// TwinCAT 3 PLC project Data
// Title: Data
// Company: TomasRompotl
// ProjectVersion: 0.0.1
// ProgramVersion: 3.1.4024.0
// libraries:
//   Base Interfaces,newest,System
//   Strings, * (TomasRompotl)
//   Tc2_System, * (Beckhoff Automation GmbH)
//   Tc2_Utilities, * (Beckhoff Automation GmbH)
// project tree:
//   Comparison/ CompareAnyType.TcPOU, ComparisonOperator.TcDUT, DataEquals.TcPOU, IsEqualAnyType.TcPOU, IsGreaterThanAnyType.TcPOU, IsGreaterThanOrEqualAnyType.TcPOU (not stored), IsLessThanAnyType.TcPOU, IsLessThanOrEqualAnyType.TcPOU, IsNotEqualAnyType.TcPOU
//   Manipulate/ ClearData.TcPOU, ClearDataAnyType.TcPOU (not stored), ShiftDataLeft.TcPOU, ShiftDataRight.TcPOU, Swap.TcPOU, SwapByPointer.TcPOU
//   QuickSort/ PartitionREAL.TcPOU (not stored), QuickSortREAL.TcPOU (not stored)
//   Sort/ SortOrder.TcTLEO, SortAnything.TcPOU (not stored), _Partition.TcPOU, _QuickSort.TcPOU
//   TableSerialization/ TableDeserializer.TcPOU, TableSerializationParameters.TcGVL (not stored), TableSerializer.TcPOU
//   Version/ Global_Version.TcGVL
// (motion and I/O tree: see PLC project types)
// real-time tasks:
//   TASK BindingTestTask: cycle T#10ms, priority 20, ADS port 350
//   TASK PlcTask: cycle T#10ms, priority 21, ADS port 351
//   TASK PlcTask1: cycle T#10ms, priority 22, ADS port 352
//   TASK PlcTask2: cycle T#10ms, priority 23, ADS port 353

// ---- Comparison/ComparisonOperator.TcDUT
{attribute 'qualified_only'}
{attribute 'strict'}
TYPE ComparisonOperator :
(
	Equal,
	NotEqual,
	LessThan,
	LessThenOrEqual,
	GreaterThan,
	GreaterThanOrEqual
);
END_TYPE

// ---- Sort/SortOrder.TcTLEO
{attribute 'qualified_only'}
{attribute 'strict'}
TYPE SortOrder :
(
	ASCENDING,
	DESCENDING
);
END_TYPE

// ---- Version/Global_Version.TcGVL
{attribute 'TcGenerated'}
{attribute 'no-analysis'}
{attribute 'linkalways'}
// This function has been automatically generated from the project information.
VAR_GLOBAL CONSTANT
	{attribute 'const_non_replaced'}
	stLibVersion_Data : ST_LibVersion := (iMajor := 0, iMinor := 0, iBuild := 1, iRevision := 0, nFlags := 0, sVersion := '0.0.1');
END_VAR

// ---- Comparison/CompareAnyType.TcPOU
FUNCTION CompareAnyType : BOOL
VAR_INPUT
	a					: __SYSTEM.AnyType; // a and b have to be same type
	is					: ComparisonOperator;
	b					: __SYSTEM.AnyType; // a and b have to be same type
END_VAR

CASE is OF
	ComparisonOperator.Equal:
		CompareAnyType := IsEqualAnyType(a, b);
	ComparisonOperator.NotEqual:
		CompareAnyType := IsNotEqualAnyType(a, b);
	ComparisonOperator.LessThan:
		CompareAnyType := IsLessThanAnyType(a, b);
	ComparisonOperator.LessThanOrEqual:
		CompareAnyType := IsLessThanOrEqualAnyType(a, b);
	ComparisonOperator.GreaterThan:
		CompareAnyType := IsGreaterThanAnyType(a, b);
	ComparisonOperator.GreaterThanOrEqual:
		CompareAnyType := IsGreaterThanOrEqualAnyType(a, b);
END_CASE

END_FUNCTION

// ---- Comparison/IsEqualAnyType.TcPOU
FUNCTION IsEqualAnyType : BOOL
VAR_INPUT
	a					: __SYSTEM.AnyType; // A and B have to be same type
	b					: __SYSTEM.AnyType; // A and B have to be same type
END_VAR

IF a.TypeClass <> b.TypeClass THEN
	RETURN;
END_IF

IsEqualAnyType := MEMCMP(a.pValue, b.pValue, TO_UDINT(a.diSize)) = 0;

END_FUNCTION

// ---- Comparison/IsNotEqualAnyType.TcPOU
FUNCTION IsNotEqualAnyType : BOOL
VAR_INPUT
	a					: __SYSTEM.AnyType; // A and B have to be same type
	b					: __SYSTEM.AnyType; // A and B have to be same type
END_VAR

IsNotEqualAnyType := NOT IsEqualAnyType(a, b);

END_FUNCTION

// ---- Comparison/IsLessThanAnyType.TcPOU
FUNCTION IsLessThanAnyType : BOOL
VAR_INPUT
	a					: __SYSTEM.AnyType; // A and B have to be same type
	b					: __SYSTEM.AnyType; // A and B have to be same type
END_VAR

IF a.TypeClass <> b.TypeClass THEN
	RETURN;
END_IF

CASE UDINT_TO_INT(a.TypeClass) OF
    IBaseLibrary.TypeClass.TYPE_BOOL :
        IsLessThanAnyType := PBOOL_TO_BOOL(a.pValue) < PBOOL_TO_BOOL(b.pValue);
    IBaseLibrary.TypeClass.TYPE_BIT :
        IsLessThanAnyType := BYTE_TO_BIT(a.pValue^) < BYTE_TO_BIT(b.pValue^);
    IBaseLibrary.TypeClass.TYPE_BYTE :
        IsLessThanAnyType := a.pValue^ < b.pValue^;
    IBaseLibrary.TypeClass.TYPE_WORD :
        IsLessThanAnyType := PWORD_TO_WORD(a.pValue) < PWORD_TO_WORD(b.pValue);
    IBaseLibrary.TypeClass.TYPE_DWORD :
        IsLessThanAnyType := PDWORD_TO_DWORD(a.pValue) < PDWORD_TO_DWORD(b.pValue);
    IBaseLibrary.TypeClass.TYPE_LWORD :
        IsLessThanAnyType := PLWORD_TO_LWORD(a.pValue) < PLWORD_TO_LWORD(b.pValue);
    IBaseLibrary.TypeClass.TYPE_SINT :
        IsLessThanAnyType := PSINT_TO_SINT(a.pValue) < PSINT_TO_SINT(b.pValue);
    IBaseLibrary.TypeClass.TYPE_INT :
        IsLessThanAnyType := PINT_TO_INT(a.pValue) < PINT_TO_INT(b.pValue);
    IBaseLibrary.TypeClass.TYPE_DINT :
        IsLessThanAnyType := PDINT_TO_DINT(a.pValue) < PDINT_TO_DINT(b.pValue);
    IBaseLibrary.TypeClass.TYPE_LINT :
        IsLessThanAnyType := PLINT_TO_LINT(a.pValue) < PLINT_TO_LINT(b.pValue);
    IBaseLibrary.TypeClass.TYPE_USINT :
        IsLessThanAnyType := PUSINT_TO_USINT(a.pValue) < PUSINT_TO_USINT(b.pValue);
    IBaseLibrary.TypeClass.TYPE_UINT :
        IsLessThanAnyType := PUINT_TO_UINT(a.pValue) < PUINT_TO_UINT(b.pValue);
    IBaseLibrary.TypeClass.TYPE_UDINT :
        IsLessThanAnyType := PUDINT_TO_UDINT(a.pValue) < PUDINT_TO_UDINT(b.pValue);
    IBaseLibrary.TypeClass.TYPE_ULINT :
        IsLessThanAnyType := PULINT_TO_ULINT(a.pValue) < PULINT_TO_ULINT(b.pValue);
    IBaseLibrary.TypeClass.TYPE_REAL :
        IsLessThanAnyType := PREAL_TO_REAL(a.pValue) < PREAL_TO_REAL(b.pValue);
    IBaseLibrary.TypeClass.TYPE_LREAL :
        IsLessThanAnyType := PLREAL_TO_LREAL(a.pValue) < PLREAL_TO_LREAL(b.pValue);
    IBaseLibrary.TypeClass.TYPE_STRING :
        IsLessThanAnyType := PSTRING_TO_STRING(a.pValue) < PSTRING_TO_STRING(b.pValue);
    IBaseLibrary.TypeClass.TYPE_TIME :
        IsLessThanAnyType := PTIME_TO_TIME(a.pValue) < PTIME_TO_TIME(b.pValue);
    IBaseLibrary.TypeClass.TYPE_DATE :
        IsLessThanAnyType := PDATE_TO_DATE(a.pValue) < PDATE_TO_DATE(b.pValue);
    IBaseLibrary.TypeClass.TYPE_DATEANDTIME :
        IsLessThanAnyType := PDT_TO_DT(a.pValue) < PDT_TO_DT(b.pValue);
    IBaseLibrary.TypeClass.TYPE_TIMEOFDAY :
        IsLessThanAnyType := PTOD_TO_TOD(a.pValue) < PTOD_TO_TOD(b.pValue);
    IBaseLibrary.TypeClass.TYPE_POINTER :
        IsLessThanAnyType := a.pValue < b.pValue;
    IBaseLibrary.TypeClass.TYPE_LTIME :
        IsLessThanAnyType := PLTIME_TO_LTIME(a.pValue) < PLTIME_TO_LTIME(b.pValue);
	ELSE
		RETURN;
END_CASE

END_FUNCTION

// ---- Comparison/IsLessThanOrEqualAnyType.TcPOU
FUNCTION IsLessThanOrEqualAnyType : BOOL
VAR_INPUT
	a					: __SYSTEM.AnyType; // A and B have to be same type
	b					: __SYSTEM.AnyType; // A and B have to be same type
END_VAR

IsLessThanOrEqualAnyType := NOT IsGreaterThanAnyType(a, b);

END_FUNCTION

// ---- Comparison/IsGreaterThanAnyType.TcPOU
FUNCTION IsGreaterThanAnyType : BOOL
VAR_INPUT
	a					: __SYSTEM.AnyType; // A and B have to be same type
	b					: __SYSTEM.AnyType; // A and B have to be same type
END_VAR

IF a.TypeClass <> b.TypeClass THEN
	RETURN;
END_IF

CASE UDINT_TO_INT(a.TypeClass) OF
    IBaseLibrary.TypeClass.TYPE_BOOL :
        IsGreaterThanAnyType := PBOOL_TO_BOOL(a.pValue) > PBOOL_TO_BOOL(b.pValue);
    IBaseLibrary.TypeClass.TYPE_BIT :
        IsGreaterThanAnyType := BYTE_TO_BIT(a.pValue^) > BYTE_TO_BIT(b.pValue^);
    IBaseLibrary.TypeClass.TYPE_BYTE :
        IsGreaterThanAnyType := a.pValue^ > b.pValue^;
    IBaseLibrary.TypeClass.TYPE_WORD :
        IsGreaterThanAnyType := PWORD_TO_WORD(a.pValue) > PWORD_TO_WORD(b.pValue);
    IBaseLibrary.TypeClass.TYPE_DWORD :
        IsGreaterThanAnyType := PDWORD_TO_DWORD(a.pValue) > PDWORD_TO_DWORD(b.pValue);
    IBaseLibrary.TypeClass.TYPE_LWORD :
        IsGreaterThanAnyType := PLWORD_TO_LWORD(a.pValue) > PLWORD_TO_LWORD(b.pValue);
    IBaseLibrary.TypeClass.TYPE_SINT :
        IsGreaterThanAnyType := PSINT_TO_SINT(a.pValue) > PSINT_TO_SINT(b.pValue);
    IBaseLibrary.TypeClass.TYPE_INT :
        IsGreaterThanAnyType := PINT_TO_INT(a.pValue) > PINT_TO_INT(b.pValue);
    IBaseLibrary.TypeClass.TYPE_DINT :
        IsGreaterThanAnyType := PDINT_TO_DINT(a.pValue) > PDINT_TO_DINT(b.pValue);
    IBaseLibrary.TypeClass.TYPE_LINT :
        IsGreaterThanAnyType := PLINT_TO_LINT(a.pValue) > PLINT_TO_LINT(b.pValue);
    IBaseLibrary.TypeClass.TYPE_USINT :
        IsGreaterThanAnyType := PUSINT_TO_USINT(a.pValue) > PUSINT_TO_USINT(b.pValue);
    IBaseLibrary.TypeClass.TYPE_UINT :
        IsGreaterThanAnyType := PUINT_TO_UINT(a.pValue) > PUINT_TO_UINT(b.pValue);
    IBaseLibrary.TypeClass.TYPE_UDINT :
        IsGreaterThanAnyType := PUDINT_TO_UDINT(a.pValue) > PUDINT_TO_UDINT(b.pValue);
    IBaseLibrary.TypeClass.TYPE_ULINT :
        IsGreaterThanAnyType := PULINT_TO_ULINT(a.pValue) > PULINT_TO_ULINT(b.pValue);
    IBaseLibrary.TypeClass.TYPE_REAL :
        IsGreaterThanAnyType := PREAL_TO_REAL(a.pValue) > PREAL_TO_REAL(b.pValue);
    IBaseLibrary.TypeClass.TYPE_LREAL :
        IsGreaterThanAnyType := PLREAL_TO_LREAL(a.pValue) > PLREAL_TO_LREAL(b.pValue);
    IBaseLibrary.TypeClass.TYPE_STRING :
        IsGreaterThanAnyType := PSTRING_TO_STRING(a.pValue) > PSTRING_TO_STRING(b.pValue);
    IBaseLibrary.TypeClass.TYPE_TIME :
        IsGreaterThanAnyType := PTIME_TO_TIME(a.pValue) > PTIME_TO_TIME(b.pValue);
    IBaseLibrary.TypeClass.TYPE_DATE :
        IsGreaterThanAnyType := PDATE_TO_DATE(a.pValue) > PDATE_TO_DATE(b.pValue);
    IBaseLibrary.TypeClass.TYPE_DATEANDTIME :
        IsGreaterThanAnyType := PDT_TO_DT(a.pValue) > PDT_TO_DT(b.pValue);
    IBaseLibrary.TypeClass.TYPE_TIMEOFDAY :
        IsGreaterThanAnyType := PTOD_TO_TOD(a.pValue) > PTOD_TO_TOD(b.pValue);
    IBaseLibrary.TypeClass.TYPE_POINTER :
        IsGreaterThanAnyType := a.pValue > b.pValue;
    IBaseLibrary.TypeClass.TYPE_LTIME :
        IsGreaterThanAnyType := PLTIME_TO_LTIME(a.pValue) > PLTIME_TO_LTIME(b.pValue);
	ELSE
		RETURN;
END_CASE

END_FUNCTION

// ---- Comparison/DataEquals.TcPOU
FUNCTION DataEquals : BOOL
VAR_INPUT
	a : ANY;
	b : ANY;
END_VAR
VAR
END_VAR

IF (a.diSize <> b.diSize) THEN
	RETURN;
END_IF

DataEquals := MEMCMP(pBuf1 := a.pValue, pBuf2 := b.pValue, n := a.diSize) = 0;

END_FUNCTION

// ---- Manipulate/ClearData.TcPOU
FUNCTION ClearData : BOOL
VAR_INPUT
	data : ANY;
END_VAR

MEMSET(destAddr := data.pValue, fillByte := 0, n := TO_UDINT(data.diSize));

END_FUNCTION

// ---- Manipulate/ShiftDataLeft.TcPOU
// Shift data from end to begin
FUNCTION ShiftDataLeft : BOOL
VAR_INPUT
	data : ANY;
	byteCount : UDINT; // How far to the left are shifted
END_VAR

MEMMOVE(destAddr := data.pValue, srcAddr := data.pValue + byteCount, n := TO_UDINT(data.diSize) - byteCount);
MEMSET(destAddr := data.pValue + TO_UDINT(data.diSize) - byteCount, fillByte := 0, n := byteCount);

END_FUNCTION

// ---- Manipulate/ShiftDataRight.TcPOU
// Shift data from end to begin
FUNCTION ShiftDataRight : BOOL
VAR_INPUT
	data : ANY;
	byteCount : UDINT; // How far to the right are shifted
END_VAR

MEMMOVE(destAddr := data.pValue + byteCount, srcAddr := data.pValue, data.diSize - byteCount);
MEMSET(destAddr := data.pValue, fillByte := 0, n := byteCount);

END_FUNCTION

// ---- Manipulate/Swap.TcPOU
// Swaps values of two variables
FUNCTION Swap
VAR_INPUT
	a : ANY;
	b : ANY;
END_VAR
VAR
	temp : POINTER TO BYTE;
END_VAR

temp := __NEW(BYTE, a.diSize);

MEMCPY(temp, a.pValue, a.diSize);
MEMCPY(a.pValue, b.pValue, a.diSize);
MEMCPY(b.pValue, temp, a.diSize);

__DELETE(temp);

END_FUNCTION

// ---- Manipulate/SwapByPointer.TcPOU
// Swaps values of two variables
FUNCTION SwapByPointer
VAR_INPUT
	a : POINTER TO BYTE;
	b : POINTER TO BYTE;
	length : DINT;
END_VAR
VAR
	temp : POINTER TO BYTE;
END_VAR

temp := __NEW(BYTE, TO_UDINT(length));

MEMCPY(temp, a, TO_UDINT(length));
MEMCPY(a, b, TO_UDINT(length));
MEMCPY(b, temp, TO_UDINT(length));

__DELETE(temp);

END_FUNCTION

// ---- Sort/_Partition.TcPOU
// Function used in QuickSort
FUNCTION _Partition : DINT
VAR_INPUT
	arr					: __SYSTEM.AnyType;
	firstElement		: __SYSTEM.AnyType;
	sortBy				: __SYSTEM.AnyType;
	memberOffset		: DWORD;
	startIndex			: DINT; // Starting comparision index
	endIndex			: DINT; // Ending comparision index
	order 				: SortOrder;
END_VAR
VAR
	pivot				: POINTER TO BYTE; // Compared number
	leftwall			: DINT; // New pivot location
	iterator			: DINT; // For iterator variable
	iterAdr				: POINTER TO BYTE;
	compA				: __SYSTEM.AnyType := sortBy; // get data of compared variable
	compB				: __SYSTEM.AnyType := sortBy;
END_VAR

pivot := arr.pValue + firstElement.diSize * endIndex;
leftwall := startIndex;

FOR iterator := startIndex TO endIndex - 1 DO

	iterAdr := arr.pValue + firstElement.diSize * iterator;
	
	compA.pValue := iterAdr + memberOffset; // data of compared variable stays the same, just point to other value
	compB.pValue := pivot + memberOffset;
	
	CASE order OF
		SortOrder.ASCENDING:
			IF (IsLessThanOrEqualAnyType(compA, compB)) THEN

				SwapByAddr(iterAdr, arr.pValue + firstElement.diSize * leftwall, firstElement.diSize);
				leftwall := leftwall + 1;
			END_IF
		SortOrder.DESCENDING:
			IF (IsGreaterThanOrEqualAnyType(compA, compB)) THEN

				SwapByAddr(iterAdr, arr.pValue + firstElement.diSize * leftwall, firstElement.diSize);
				leftwall := leftwall + 1;
			END_IF
	END_CASE
END_FOR

SwapByAddr(arr.pValue + firstElement.diSize * leftwall, pivot, firstElement.diSize);

_Partition := leftwall;

END_FUNCTION

// ---- Sort/_QuickSort.TcPOU

FUNCTION _QuickSort
VAR_INPUT
	Arr					: __SYSTEM.AnyType;
	FirstElement		: __SYSTEM.AnyType;
	SortBy				: __SYSTEM.AnyType;
	MemberOffset		: DWORD;
	StartIndex			: DINT; // Start index
	EndIndex			: DINT; // End index
	Order 				: SortOrder;
END_VAR
VAR 
	PivotIndex			: DINT; // Partitioning point
END_VAR


IF StartIndex < EndIndex THEN

	PivotIndex := _Partition(Arr, FirstElement, SortBy, MemberOffset, StartIndex, EndIndex, Order);
	_QuickSort(Arr, FirstElement, SortBy, MemberOffset, StartIndex, PivotIndex - 1, Order);
	_QuickSort(Arr, FirstElement, SortBy, MemberOffset, PivotIndex + 1, EndIndex, Order);
END_IF

END_FUNCTION

// ---- TableSerialization/TableDeserializer.TcPOU
FUNCTION_BLOCK TableDeserializer
VAR
	_DataString : POINTER TO STRING;
	dataLength : DINT;
	rowDefinition : __SYSTEM.AnyType;
	_RowCount : DINT;
	_ColumnDefinitionBuffer : ARRAY[0..MaxColumnCount - 1] OF __SYSTEM.AnyType;
	_ColumnNameBuffer : ARRAY[0..MaxColumnCount - 1] OF T_MaxString;
	columnNamesOutput : __SYSTEM.AnyType;
	definedColumns : INT;

	_Separator : STRING := ',';
	_NewLine : STRING := '$N'; // Default is Windows newline.
	_DecimalSeparator : STRING := '.';
END_VAR
VAR CONSTANT
	MaxColumnCount : INT := TableSerializationParameters.DeserializerMaxColumns;
	DefaultDecimalSeparator : STRING := '.';
END_VAR

{attribute 'monitoring' := 'call'}
PROPERTY DataString : POINTER TO STRING
GET
DataString := _DataString;
END_GET
SET
_DataString := DataString;
END_SET
END_PROPERTY

{attribute 'monitoring' := 'call'}
PROPERTY DecimalSeparator : STRING
GET
DecimalSeparator := _DecimalSeparator;
END_GET
SET
_DecimalSeparator := DecimalSeparator;
END_SET
END_PROPERTY

METHOD DefineColumnNamesOutput : REFERENCE TO TableDeserializer
VAR_INPUT
	columnNames : ANY; 
END_VAR
columnNamesOutput := columnNames;

DefineColumnNamesOutput REF= THIS^;
END_METHOD

METHOD DefineNextColumn : REFERENCE TO TableDeserializer
VAR_INPUT
	columnInFirstRow : ANY; 
END_VAR
IF (definedColumns < MaxColumnCount) THEN
	_ColumnDefinitionBuffer[definedColumns] := columnInFirstRow;
	definedColumns := definedColumns + 1;
END_IF

DefineNextColumn REF= THIS^;
END_METHOD

METHOD DefineRow : REFERENCE TO TableDeserializer
VAR_INPUT
	firstRow : ANY;
END_VAR
rowDefinition := firstRow;

DefineRow REF= THIS^;
END_METHOD

METHOD Deserialize : DINT
VAR_INPUT
	includingHeader : BOOL;
END_VAR
VAR
	caret : DINT;
END_VAR
dataLength := LEN2(dataString);
IF (includingHeader) THEN
	caret := ReadHeader();
END_IF
caret := ReadAllRows(caret);

Deserialize := caret;
END_METHOD

{attribute 'monitoring' := 'call'}
PROPERTY NewLine : STRING
GET
NewLine := _NewLine;
END_GET
SET
_NewLine := NewLine;
END_SET
END_PROPERTY

METHOD PRIVATE ReadAllRows : DINT
VAR_INPUT
	startCaret : DINT;
END_VAR
VAR
	caret : DINT;
	i : DINT;
END_VAR
caret := startCaret;

FOR i := 0 TO _RowCount - 1 DO
	IF (caret >= dataLength) THEN
		EXIT;
	END_IF
	caret := ReadRow(i, caret);
END_FOR

ReadAllRows := caret;
END_METHOD

METHOD PRIVATE ReadHeader : DINT
VAR
	i : DINT;
	
	caret : DINT;
	lineEnd : DINT;
	cellLength : DINT;
	
	cell : T_MaxString;
END_VAR
ClearData(_ColumnNameBuffer);

lineEnd := FIND2(pSrcString := _DataString, pFindString := ADR(_NewLine));
IF (lineEnd = 0) THEN
	lineEnd := dataLength;
END_IF

FOR i := 0 TO definedColumns - 1 DO
	cellLength := FIND2(pSrcString := _DataString + caret, pFindString := ADR(_Separator));
	IF (caret + cellLength > lineEnd) THEN
		cellLength := lineEnd - caret;
	END_IF
	IF (cellLength = 0) THEN
		cellLength := lineEnd;
	END_IF

	MEMSET(destAddr := ADR(cell), fillByte := 0, n := SIZEOF(cell));
	MEMCPY(destAddr := ADR(cell), srcAddr := _DataString + caret, n := MIN(SIZEOF(cell) - 1, cellLength - 1));
	StringToAny(cell, _ColumnNameBuffer[i]);
	
	IF (cellLength = dataLength) THEN
		caret := lineEnd;
	ELSIF (cellLength = lineEnd) THEN
		caret := lineEnd;
	ELSE
		caret := caret + cellLength;
	END_IF
END_FOR

MEMCPY(
	destAddr := columnNamesOutput.pValue,
	srcAddr := ADR(_ColumnNameBuffer),
	n := MIN(columnNamesOutput.diSize, SIZEOF(_ColumnNameBuffer))
);

ReadHeader := caret;
END_METHOD

METHOD PRIVATE ReadRow : DINT
VAR_INPUT
	row : DINT;
	startCaret : DINT;
END_VAR
VAR
	i : DINT;
	
	caret : DINT;
	lineLength : DINT;
	cellLength : DINT;
	
	cell : T_MaxString;
	
	tableCell : __SYSTEM.AnyType;
END_VAR
caret := startCaret;

lineLength := FIND2(pSrcString := _DataString + caret, pFindString := ADR(_NewLine));
IF (lineLength = 0) THEN
	lineLength := dataLength;
END_IF

FOR i := 0 TO definedColumns - 1 DO
  IF (caret >= dataLength) THEN
		EXIT;
	END_IF
	cellLength := FIND2(pSrcString := _DataString + caret, pFindString := ADR(_Separator));
	IF (cellLength = 0 OR caret + cellLength > startCaret + lineLength) THEN
		cellLength := lineLength + startCaret - caret;
	END_IF
	IF (cellLength = 0) THEN
		caret := dataLength;
		EXIT;
	END_IF

	ClearData(cell);
	MEMCPY(destAddr := ADR(cell), srcAddr := _DataString + caret, n := MIN(SIZEOF(cell) - 1, cellLength - 1));
	tableCell := _ColumnDefinitionBuffer[i];
	tableCell.pValue := tableCell.pValue + rowDefinition.diSize * row;
	CASE tableCell.TypeClass OF
		TYPE_REAL, TYPE_LREAL:
			ReplaceString(cell, _DecimalSeparator, DefaultDecimalSeparator);
	END_CASE
	StringToAnyType(cell, tableCell);
	
	IF (cellLength = dataLength) THEN
		caret := startCaret + lineLength;
	ELSIF (cellLength = lineLength) THEN
		caret := startCaret + lineLength;
	ELSE
		caret := caret + cellLength;
	END_IF
END_FOR

ReadRow := caret;
END_METHOD

{attribute 'monitoring' := 'call'}
PROPERTY RowCount : DINT
GET
RowCount := _RowCount;
END_GET
SET
_RowCount := RowCount;
END_SET
END_PROPERTY

{attribute 'monitoring' := 'call'}
PROPERTY Separator : STRING
GET
Separator := _Separator;
END_GET
SET
_Separator := Separator;
END_SET
END_PROPERTY

END_FUNCTION_BLOCK

// ---- TableSerialization/TableSerializer.TcPOU
FUNCTION_BLOCK TableSerializer
VAR
	_StringBuilder : REFERENCE TO StringBuilderExtBuffer;
	
	rowDefinition : __SYSTEM.AnyType;
	_RowCount : DINT;
	_ColumnDefinitionBuffer : ARRAY[0..MaxColumnCount - 1] OF __SYSTEM.AnyType;
	_ColumnNameBuffer : ARRAY[0..MaxColumnCount - 1] OF T_MaxString;
	definedColumns : INT;
	
	_Separator : STRING := ','; // Default separator ';' is compatible with european decimal separator '.'.
	_NewLine : STRING := '$N'; // Default is Windows newline.
	_DecimalSeparator : STRING := '.';
END_VAR
VAR CONSTANT
	MaxColumnCount : INT := TableSerializationParameters.SerializerMaxColumns;
	DefaultDecimalSeparator : STRING := '.';
END_VAR

METHOD PRIVATE AddColumnHeader
VAR
	column : INT;
END_VAR
FOR column := 0 TO definedColumns - 1 DO
	IF (column > 0) THEN
		_StringBuilder.Append(_Separator);
	END_IF
	
	_StringBuilder.Append(_ColumnNameBuffer[column]);
END_FOR
END_METHOD

METHOD PRIVATE AddLine
VAR_INPUT
	rowIndex : DINT;
END_VAR
VAR
	column : INT;
	currentData : __SYSTEM.AnyType;
	converted : T_MaxString;
END_VAR
FOR column := 0 TO definedColumns - 1 DO
	IF (column > 0) THEN
		_StringBuilder.Append(_Separator);
	END_IF
	
	currentData := _ColumnDefinitionBuffer[column];
	currentData.pValue := rowDefinition.pValue + (rowDefinition.diSize * rowIndex) + (currentData.pValue - rowDefinition.pValue);
	
	IF (currentData.TypeClass = IBaseLibrary.TypeClass.TYPE_STRING) THEN
		_StringBuilder.AppendByPointer(currentData.pValue);
	ELSE
		converted := AnyTypeToString(currentData);
		
		CASE currentData.TypeClass OF
			TYPE_REAL, TYPE_LREAL:
				ReplaceString(converted, DefaultDecimalSeparator, _DecimalSeparator);
		END_CASE
		
		_StringBuilder.Append(converted);
	END_IF
END_FOR
END_METHOD

METHOD PRIVATE AddNewLine
_StringBuilder.Append(_NewLine);
END_METHOD

METHOD PRIVATE AddRows
VAR
	row : DINT;
END_VAR
FOR row := 0 TO _RowCount - 1 DO
	IF (row > 0) THEN
		AddNewLine();
	END_IF
	AddLine(row);
END_FOR
END_METHOD

{attribute 'monitoring' := 'call'}
PROPERTY DecimalSeparator : STRING
GET
DecimalSeparator := _DecimalSeparator;
END_GET
SET
_DecimalSeparator := DecimalSeparator;
END_SET
END_PROPERTY

METHOD DefineNextColumn : REFERENCE TO TableSerializer
VAR_INPUT
	columnInFirstRow : ANY; 
END_VAR
IF (definedColumns < MaxColumnCount) THEN
	_ColumnDefinitionBuffer[definedColumns] := columnInFirstRow;
	definedColumns := definedColumns + 1;
END_IF

DefineNextColumn REF= THIS^;
END_METHOD

METHOD DefineNextColumnWithName : REFERENCE TO TableSerializer
VAR_INPUT
	columnInFirstRow : ANY;
	name : T_MaxString;
END_VAR
IF (definedColumns < MaxColumnCount) THEN
	_ColumnDefinitionBuffer[definedColumns] := columnInFirstRow;
	_ColumnNameBuffer[definedColumns] := name;
	definedColumns := definedColumns + 1;
END_IF

DefineNextColumnWithName REF= THIS^;
END_METHOD

METHOD DefineRow : REFERENCE TO TableSerializer
VAR_INPUT
	firstRow : ANY;
END_VAR
rowDefinition := firstRow;

DefineRow REF= THIS^;
END_METHOD

{attribute 'monitoring' := 'call'}
PROPERTY NewLine : STRING
GET
NewLine := _NewLine;
END_GET
SET
_NewLine := NewLine;
END_SET
END_PROPERTY

{attribute 'monitoring' := 'call'}
PROPERTY RowCount : DINT
GET
RowCount := _RowCount;
END_GET
SET
_RowCount := RowCount;
END_SET
END_PROPERTY

{attribute 'monitoring' := 'call'}
PROPERTY Separator : STRING
GET
Separator := _Separator;
END_GET
SET
_Separator := Separator;
END_SET
END_PROPERTY

METHOD Serialize
VAR_INPUT
	includeHeader : BOOL;
	clearBuffer : BOOL;
END_VAR
IF (clearBuffer) THEN
	_StringBuilder.Clear();
END_IF
IF (includeHeader) THEN
	AddColumnHeader();
	AddNewLine();
END_IF
AddRows();
END_METHOD

{attribute 'monitoring' := 'call'}
PROPERTY SerializedLength : DINT
GET
SerializedLength := _StringBuilder.Length;
END_GET
END_PROPERTY

{attribute 'monitoring' := 'call'}
PROPERTY SerializedString : POINTER TO STRING
GET
SerializedString := stringBuilder.BufferRef.pValue;
END_GET
END_PROPERTY

{attribute 'monitoring' := 'call'}
PROPERTY StringBuilder : REFERENCE TO StringBuilderExtBuffer
GET
StringBuilder REF= _StringBuilder;
END_GET
SET
_StringBuilder REF= StringBuilder;
END_SET
END_PROPERTY

END_FUNCTION_BLOCK
